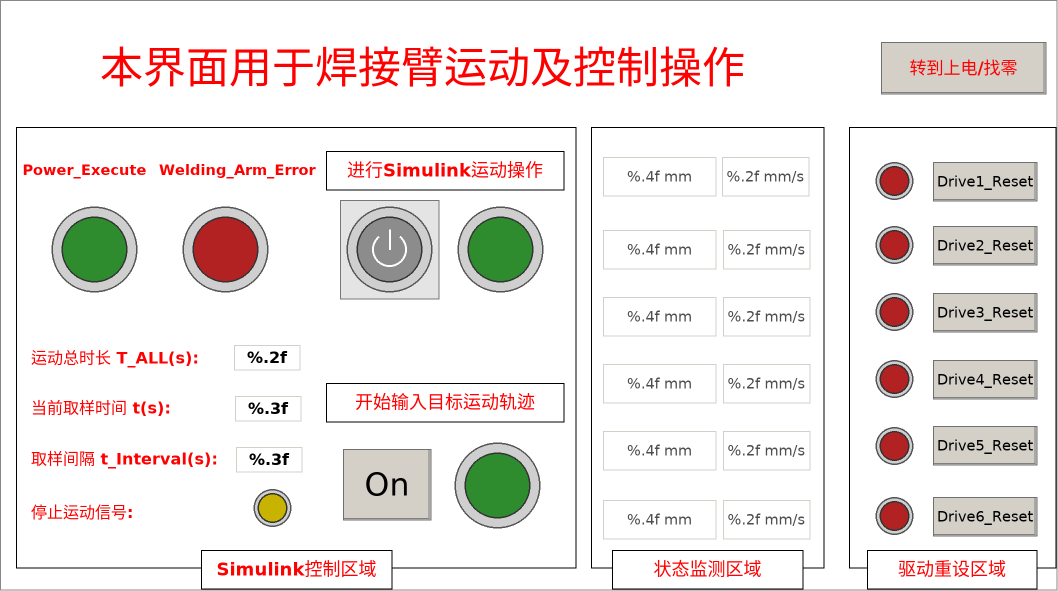
VISUALIZATION Visu_Welding_Arm_SimulinkMove  // 1058x591
    Rectangle (849,127 207x441)
    Rectangle (16,127 560x441)
    Label (19,154 131x32), "Power_Execute"
    Label (160,154 155x32), "Welding_Arm_Error"
    RoundedRectangle (326,151 238x39), "进行Simulink运动操作"
    Lamp1 (451,199 99x101), variable: Welding_Arm_Movement.ExSetPoint_Execute, style: Lamp-Lamp1-Green
    PowerSwitch (340,199 99x101), variable: Welding_Arm_Movement.ExSetPoint_Execute, behaviour: TOGGLE, style: Switch-PowerSwitch-Gray
    Lamp1 (867,159 55x44), variable: Welding_Arm_Control.Axis_Error[1], style: Lamp-Lamp1-Red
    Button (933,162 104x39), "Drive1_Reset"
        toggle Welding_Arm_Control.Axis_Reset[1]
    Lamp1 (867,223 55x44), variable: Welding_Arm_Control.Axis_Error[2], style: Lamp-Lamp1-Red
    Button (933,226 104x39), "Drive2_Reset"
        toggle Welding_Arm_Control.Axis_Reset[2]
    Lamp1 (867,290 55x44), variable: Welding_Arm_Control.Axis_Error[3], style: Lamp-Lamp1-Red
    Button (933,293 104x39), "Drive3_Reset"
        toggle Welding_Arm_Control.Axis_Reset[3]
    Lamp1 (867,357 55x44), variable: Welding_Arm_Control.Axis_Error[4], style: Lamp-Lamp1-Red
    Button (933,360 104x39), "Drive4_Reset"
        toggle Welding_Arm_Control.Axis_Reset[4]
    Lamp1 (867,424 55x44), variable: Welding_Arm_Control.Axis_Error[5], style: Lamp-Lamp1-Red
    Button (933,426 104x39), "Drive5_Reset"
        toggle Welding_Arm_Control.Axis_Reset[5]
    Lamp1 (867,494 55x44), variable: Welding_Arm_Control.Axis_Error[6], style: Lamp-Lamp1-Red
    Button (933,497 104x39), "Drive6_Reset"
        toggle Welding_Arm_Control.Axis_Reset[6]
    Textfield (235,396 66x25), "%.3f", text variable: Welding_Arm_Movement.t
    Label (28,396 188x24), "当前取样时间 t(s):"
    Lamp1 (245,486 55x44), variable: Welding_Arm_Movement.ExtSetPointDisable, style: Lamp-Lamp1-Yellow
    Label (28,499 182x27), "停止运动信号:"
    Label (28,447 205x24), "取样间隔 t_Interval(s):"
    Textfield (236,447 66x25), "%.3f", text variable: Welding_Arm_Movement.t_Interval
        OnMouseClick: write Welding_Arm_Movement.t_Interval via Default
    Label (28,346 199x24), "运动总时长 T_ALL(s):"
    Textfield (234,345 66x25), "%.2f", text variable: Welding_Arm_Movement.T_ALL
    RoundedRectangle (326,383 238x39), "开始输入目标运动轨迹"
    Lamp1 (448,435 99x101), variable: Welding_Arm_Movement.ExtSetPointEnable, style: Lamp-Lamp1-Green
    Button (343,449 88x71), "On"
        toggle Welding_Arm_Movement.ExtSetPointEnable
    Button (881,42 165x52), "转到上电/找零"
        OnMouseClick: change screen: Visu_Welding_Arm_Power
    Lamp1 (176,199 99x101), variable: Welding_Arm_Control.Welding_Arm_Error, style: Lamp-Lamp1-Red
    Lamp1 (45,199 99x101), variable: Welding_Arm_Control.Power_Execute, style: Lamp-Lamp1-Green
    Label (16,38 813x60), "本界面用于焊接臂运动及控制操作"
    RoundedRectangle (201,550 191x39), "Simulink控制区域"
    Rectangle (591,127 233x441)
    Textfield (603,157 113x39), "%.4f mm", text variable: Welding_Arm_Control.Axis_ActPostion[1]
    Textfield (722,157 87x39), "%.2f mm/s", text variable: Welding_Arm_Control.Axis_ActVelocity[1]
    Textfield (603,230 113x39), "%.4f mm", text variable: Welding_Arm_Control.Axis_ActPostion[2]
    Textfield (723,230 87x39), "%.2f mm/s", text variable: Welding_Arm_Control.Axis_ActVelocity[2]
    Textfield (603,297 113x39), "%.4f mm", text variable: Welding_Arm_Control.Axis_ActPostion[3]
    Textfield (723,297 87x39), "%.2f mm/s", text variable: Welding_Arm_Control.Axis_ActVelocity[3]
    Textfield (603,364 113x39), "%.4f mm", text variable: Welding_Arm_Control.Axis_ActPostion[4]
    Textfield (723,364 87x39), "%.2f mm/s", text variable: Welding_Arm_Control.Axis_ActVelocity[4]
    Textfield (603,431 113x39), "%.4f mm", text variable: Welding_Arm_Control.Axis_ActPostion[5]
    Textfield (723,431 87x39), "%.2f mm/s", text variable: Welding_Arm_Control.Axis_ActVelocity[5]
    Textfield (603,500 113x39), "%.4f mm", text variable: Welding_Arm_Control.Axis_ActPostion[6]
    Textfield (723,500 87x39), "%.2f mm/s", text variable: Welding_Arm_Control.Axis_ActVelocity[6]
    RoundedRectangle (612,550 191x39), "状态监测区域"
    RoundedRectangle (867,550 170x39), "驱动重设区域"
END_VISUALIZATION

(* stored: Version 1.1.0.1, ProductVersion 3.1.4020.12
   Visu Visu_Welding_Arm_SimulinkMove: Id {6eaba7fa-d490-4a44-8849-d266ab04451b} *)
